// TIA Portal V16 export
// export: Created 2021-07-12T14:47:18.8495622Z, ExportSetting WithDefaults, DisplayName Totally Integrated Automation Portal, DisplayVersion V16, DisplayName TIA Portal Version Control Interface, DisplayVersion V16, DisplayName TIA Portal Openness, DisplayVersion V16, DisplayName STEP 7 Professional, DisplayVersion V16, DisplayName STEP 7 Safety, DisplayVersion V16, DisplayName WinCC Professional, DisplayVersion V16
TYPE "LSimaHydTO_typeProfile"
TITLE = LSimaHydTO_typeProfile
// Configuration for the profile point
// stored: IsFailsafeCompliant false
   STRUCT
      LeadingValue { S7_SetPoint := 'True'} : Array[0.."LSIMAHYD_PROFILE_POINTS_UPPER_LIMIT"] of Real;   // Input values array
      Value { S7_SetPoint := 'True'} : Array[0.."LSIMAHYD_PROFILE_POINTS_UPPER_LIMIT"] of Real;   // Output values array
      MaxIdx { S7_SetPoint := 'True'} : Int;   // Max used index in arrays
   END_STRUCT;
END_TYPE
